TYPE ST_AlarmTags :
STRUCT
	AlarmID: ARRAY [1..NO_OF_ALARM_TAG] OF BOOL;
END_STRUCT
END_TYPE

(* stored: Version 1.1.0.1, ProductVersion 3.1.4022.12
   DUT ST_AlarmTags: Id {ac2cb686-f98a-46dd-8842-64254e4b96c0} *)
